PROGRAM main
  VAR
    LocalVar0 : BOOL;
    LocalVar1 : BOOL;
    LocalOut0 : BOOL;
    LocalOut1 : BOOL;
  END_VAR

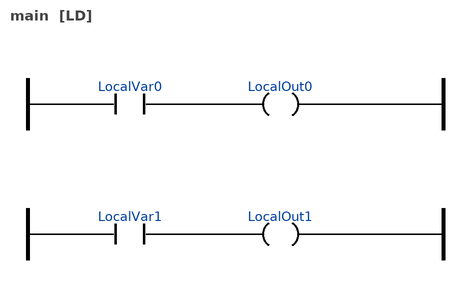
(* LD diagram, written out as Structured Text *)
LocalOut0 := LocalVar0;
LocalOut1 := LocalVar1;
END_PROGRAM
